{attribute 'linkalways'} 
{attribute 'no_explicit_call' := 'This FB is a CLASS and must be accessed using methods or properties'}
{attribute 'enable_dynamic_creation'}
FUNCTION_BLOCK FINAL NE_LREAL EXTENDS Node
VAR
	in1 : _LREAL(0.0);
	in2 : _LREAL(0.0);
	out : _BOOL(FALSE);
END_VAR

METHOD PUBLIC Clone : I_Node
VAR
	pNode : POINTER TO NE_LREAL;
END_VAR
pNode := __NEW(NE_LREAL);
Clone := pNode^;
END_METHOD

METHOD FB_init : BOOL
VAR_INPUT
	bInitRetains : BOOL; // if TRUE, the retain variables are initialized (warm start / cold start)
	bInCopyCode : BOOL;  // if TRUE, the instance afterwards gets moved into the copy code (online change)
END_VAR
AddInput('in1',THIS^.in1);
AddInput('in2',THIS^.in2);
AddOutput('out', THIS^.out);
END_METHOD

METHOD PROTECTED OnExecute
VAR
END_VAR
out.Value := in1.Value <> in2.Value;
END_METHOD

END_FUNCTION_BLOCK

(* stored: Version 1.1.0.1, ProductVersion 3.1.4024.15
   POU NE_LREAL: Id {cfda67b8-44ae-4d64-9a17-6bbcb7956e89}, SpecialFunc None
   Folder Constructor: Id {f9067226-368f-472b-8ad2-6c3e7c11fe5c}
   Method Clone: Id {763a7058-3d0a-4d25-870d-2052081fc71b}
   Method FB_init: Id {6a9caa58-e305-4cd8-ad8a-a901bfc2d16e}
   Method OnExecute: Id {d45c27ed-736d-43bc-a781-0ecb17fb2b79} *)
